(*======================================================================================================================================*)
(*fb_RS485FiFoMaster:	Einfaches Senden eines Telegrams über RS485*)
(*
Date          	| Version    	| created under        	| Author          	| Remark *)
(*====================================================================================================================================================*)
(*10/05/2025   	| 1.00      		| TC3		  		| N.Kersting       | first release *)
(*10/05/2025   	| 1.01      		| TC3		  		| N.Kersting       | Nun wird der Empfang auch mit Implementiert  *)
(*13/05/2025   	| 1.02      		| TC3		  		| N.Kersting       | Busbelastungstest Implementiert - Sendet Durchgehend Strings *)
(*14/05/2025   	| 1.03      		| TC3		  		| N.Kersting       | Busauslastung direkt Implementiert *)
(*====================================================================================================================================================*)
FUNCTION_BLOCK fb_RS485FiFoMaster_1
VAR_INPUT
	I_sSendCmdFiFo				:ARRAY[1..cMaxRS485CMDFiFo] OF STRING(255);
	I_bExecute					:BOOL := TRUE;
	I_bBusBelastungstest		:BOOL;
	I_bReset					:BOOL;
	I_pTxBuffer					:POINTER TO ComBuffer;  (*Zeiger auf TX-Buffer*)
	I_pRxBuffer   				:POINTER TO ComBuffer;  (*Zeiger auf RX-Buffer*)
END_VAR
VAR_OUTPUT
	Q_sReceiveString			:STRING(255);		
	Q_lrBusAuslastung			:LREAL;
	Q_bBusy						:BOOL;
	Q_bDone						:BOOL;
	Q_bError					:BOOL;
	Q_sState					:STRING;
	Q_stStates					:ST_FiFoMaster_State;
END_VAR
VAR
	bFirstCycle					:BOOL := TRUE;
	tVerzReceive				:TIME := T#30MS;			(* Zeit, die zum Empfangen bleibt *)
	
	tonSend						:ton;
	fbSend     					:SendString255;
	fbReceive   				:ReceiveString255;
	sStartZeichen				:BYTE := 16#FD;				(* Startzeichen Präfix *)
	sEndZeichen					:BYTE := 16#FE;				(* Endzeichen Suffix *)
	sReceivedMEMString			:STRING(255);
	sReceivedString				:STRING(255);
	iStep						:INT;
	iStepReceive				:INT;
	iMaxBufferBlocking			:INT := 0;
	bBusyMem					:BOOL;
	sStep						:STRING;
	sString						:STRING(255);
	sStringSend					:STRING(255);
	tonVerzReceive				:ton;	
	tonTimeout					:ton;
	bStringSend					:BOOL := FALSE;
	icntError					:INT;
	
	iFiFoRow					:INT := 1;
	icntFiFo					:INT;
	i,h							:INT;
	iStepFiFo					:INT;
	
	bBusBelastungstest			:BOOL := FALSE;
	bBusAuslastung				:BOOL := TRUE;
	fbBusAuslastung				:fb_FilterArray;
END_VAR

(*============================================================================================*)
tonTimeout(
	PT:=T#1S);
	
tonVerzReceive(
	pt := tVerzReceive);

(* Busbelastungstest *)	
bBusBelastungstest := I_bBusBelastungstest;

sReceivedMEMString:='';
(*============================================================================================*)	
icntFiFo := 0;
FOR i := 1 TO cMaxRS485CMDFiFo BY 1 DO 
	IF (I_sSendCmdFiFo[i]<> '')
	THEN
		icntFiFo := icntFiFo +1;
	END_IF
END_FOR

(*============================================================================================*)
CASE iStepFiFo OF
-1:	sStep := 'FiFo INIT';
	bFirstCycle := FALSE;
	Q_bBusy := FALSE;
	iFiFoRow := 1;
	
	FOR h := 1 TO cMaxRS485CMDFiFo BY 1 DO
		GVL_RS485FiFoSend.bSendDoneFiFo[h] :=TRUE;
	END_FOR
	
	iStepFiFo := 0;

(*============================================================================================*)
0:	sStep := 'Warten, dass FiFo gefüllt wird';
	iFiFoRow := 1;
	bStringSend := FALSE;
	Q_bBusy := FALSE;
	tonVerzReceive.IN := (I_pTxBuffer^.Count<= INT_TO_UINT(iMaxBufferBlocking));
	
	IF (icntFiFo > 0
		OR  bBusBelastungstest)
		AND NOT bFirstCycle
		AND NOT fbReceive.StringReceived
		AND tonVerzReceive.Q
	THEN
		Q_bBusy := TRUE;
		iStepFiFo := 1;
	ELSIF
		bFirstCycle
	THEN
		iStepFiFo := -1;
	END_IF
	
(*============================================================================================*)	
1:	sStep := 'Prüfen ob STRING in FiFo Zeile gefüllt*';
	sStringSend :=	I_sSendCmdFiFo[iFiFoRow]; 
	
	(* Prüfen ob in der ausgewählten Zeile etwas steht *)
	IF I_sSendCmdFiFo[iFiFoRow] = ''
	THEN
		IF iFiFoRow < cMaxRS485CMDFiFo
		THEN
			iFiFoRow := iFiFoRow+1; (* Nächste Zeile, bis etwas drin Steht *)
		ELSE
			IF bBusBelastungstest
			THEN
				sStringSend :=	CONCAT(F_ToCHR(sStartZeichen),'ServiceTOOL-BUSBELASTUNGSTEST-BURSTFIREMODE');
				sStringSend :=	CONCAT(sStringSend,F_ToCHR(sEndZeichen));
				(* Senden *)
				
				IF NOT I_pTxBuffer^.blocked
					AND (I_pTxBuffer^.Error=0)
					AND NOT fbReceive.StringReceived
				THEN
					sStep := 'Prüfe ob Senden noch aktiv ist';
					bStringSend := TRUE;
					sString :=	sStringSend;
					Q_bDone := FALSE;
					Q_bError := FALSE;
					iStepFiFo := iStepFiFo+1;
				END_IF
			ELSE
				iStepFiFo := 0;	(* Alle Zeilen Abgearbeitet *)
			END_IF
			
		END_IF
	ELSE
		(* Senden *)
		GVL_RS485FiFoSend.bSendDoneFiFo[iFiFoRow] :=FALSE;
		
		IF NOT I_pTxBuffer^.blocked
			AND (I_pTxBuffer^.Error=0)
			AND NOT fbReceive.StringReceived
		THEN
			sStep := 'Prüfe ob Senden noch aktiv ist';
			bStringSend := TRUE;
			sString :=	sStringSend;
			Q_bDone := FALSE;
			Q_bError := FALSE;
			iStepFiFo := iStepFiFo+1;
		END_IF
	END_IF
	
(*============================================================================================*)		
2:	sStep := 'Starte Senden';
	Q_bBusy := TRUE;
	tonTimeout.IN := fbSend.Busy;
	
	IF NOT fbSend.Busy
		AND NOT fbReceive.StringReceived
	THEN
		tonSend.IN := FALSE;
		bStringSend := FALSE;
		iStepFiFo := iStepFiFo+1;
	ELSIF
		(fbSend.Error >0)
		AND NOT (fbSend.Error = 2)
	THEN
		sStep := CONCAT('ERROR-',sStep);
		sStep := CONCAT(sStep,'- ');
		sStep := CONCAT(sStep,INT_TO_STRING(fbSend.Error));
		iStepFiFo := -2;
	ELSIF
		tonTimeout.Q
	THEN
		sStep := CONCAT('ERROR- Timeout',sStep);
		iStepFiFo := -2;
	END_IF

3:	(* Senden*)		
	GVL_RS485FiFoSend.bSendDoneFiFo[iFiFoRow] :=TRUE;
	
	IF iFiFoRow < iFiFoRow
	THEN
		iFiFoRow := iFiFoRow+1;
		iStepFiFo := 1;
	ELSE
		Q_bDone := TRUE;
		iStepFiFo := 0;
	END_IF

ELSE
(*============================================================================================*)
	Q_bError := TRUE;
	Q_bBusy := FALSE;
	bBusyMem := FALSE;
	tonTimeout.IN := FALSE;
	
	IF I_bReset
	THEN
		iStepFiFo := 0;
	END_IF
END_CASE

IF bStringSend
THEN
	fbSend(
		SendString:= 	sString,
		TXbuffer:= 		I_pTxBuffer^);
ELSE
	(* Empfangen *)
	ac00_Receive();
END_IF

(* Empfangsmerker 0 Setzen am ende Eines Zyklus *)
Q_sReceiveString := sReceivedMEMString;

(* Busauslastung tracken*)
ac99_Diagnose();

Q_sState :=	sStep;

(* StatusStruktur für Visu *)
Q_stStates.bBusy				:=	Q_bBusy;
Q_stStates.bDone				:=	Q_bDone;
Q_stStates.bError				:=	Q_bError;
Q_stStates.iFiFoCount			:=	icntFiFo;
Q_stStates.iFiFoRow				:=	iFiFoRow;
Q_stStates.lrBusAuslastung		:=	Q_lrBusAuslastung;
Q_stStates.sReceiveString 		:=	Q_sReceiveString;
Q_stStates.sSendString 			:=	sString;
Q_stStates.sState 				:=	Q_sState;

ACTION ac00_Receive:
(* Empfangen *)
CASE iStepReceive OF		
0:	fbReceive(
		Prefix := 			F_ToCHR(sStartZeichen),
		Suffix := 			F_ToCHR(sEndZeichen),
		Timeout:= , 
		Reset:= , 
		StringReceived=> , 
		Busy=> , 
		Error=> , 
		RxTimeout=> , 
		ReceivedString:= 	sReceivedString, 
		RXbuffer:= 			I_pRxBuffer^);
		
	IF fbReceive.StringReceived
	THEN
		iStepReceive := 1;
		sReceivedMEMString := sReceivedString;
	END_IF
	
1:	sReceivedString := '';
	iStepReceive := 0;
	
END_CASE
END_ACTION

ACTION ac99_Diagnose:
(* Busauslastung Prüfen *)
fbBusAuslastung(
	I_bExcecute:= 	bBusAuslastung, 
	I_nWert:= 		UINT_TO_LREAL(I_pTxBuffer^.Count), 
	I_nFilterWert:= 50, 
	Q_nFilter=> 	Q_lrBusAuslastung);
END_ACTION

END_FUNCTION_BLOCK

(* stored: Version 1.1.0.1, ProductVersion 3.1.4024.12
   POU fb_RS485FiFoMaster_1: Id {43d01709-2e2b-4911-9e8e-f4afe5c1d365}, SpecialFunc None
   Action ac00_Receive: Id {d4193227-78e7-496f-a95e-8c86dd0bf4cd}
   Action ac99_Diagnose: Id {2012345a-2ad6-4c53-b270-1165c6c4e821} *)
